(* IEC 61131-3 sources: Structured-Text/Source Code/Auxiliary/SCP_ST, 2 files *)

(* ---- Local Variables.ST ---- *)
VAR_INPUT
	Input:	DINT;
	InMin:	REAL;
	InMax:	REAL;
	OutMin:	REAL;
	OutMax: REAL;
END_VAR

VAR_OUTPUT
	Output:	INT;
END_VAR

VAR
	Temp:	REAL;
END_VAR

(* ---- SCP_ST.ST ---- *)
//Scale with Parameters//
//Paul Atkins, 05/02/2021//

//Enforce Range Limits//
IF ANY_TO_REAL(Input) < InMin THEN
	Temp := InMin;
ELSIF ANY_TO_REAL(Input) > InMax THEN
	Temp := InMax;
ELSE
	Temp := ANY_TO_REAL(Input);
END_IF;

//Scale input and map to output//
Output := ANY_TO_INT(	(Temp - InMin) / (InMax - InMin) * (OutMax - OutMin) + OutMin	);
